{attribute addProperty BoxType "EP3314-0002-0016"}
{attribute addProperty Id "TC_TCInputs_ChannelAT %I*ARRAY[0..3] OF TC_TCInputs_Channel_4364CDB6296370WcStateAT %I*WcState_F855686C1620InfoDataAT %I*InfoData_BC63D37F80100"}
{attribute addProperty CRC "3890804559"}
{attribute addProperty SizeInBites "392"}
{attribute addProperty SizeInBytes "49"}
TYPE EP3314_77584909 :
STRUCT
	{attribute addProperty Name "TC_TCInputs_Channel"}
	TC_TCInputs_Channel : ARRAY[0..3] OF TC_TCInputs_Channel_4364CDB6;
	{attribute addProperty Name "WcState"}
	WcState : WcState_F855686C;
	{attribute addProperty Name "InfoData"}
	InfoData : InfoData_BC63D37F;
END_STRUCT
END_TYPE

(* stored: Version 1.2.0.0, ProductVersion 3.1.4024.9
   DUT EP3314_77584909: Id {3ade7508-9549-4548-b31a-b5ef27b3cd4e} *)
